# EPICS autosave request: ADApp/Db/marCCD_settings.req
$(P)$(R)ReadTiffTimeout
